// TIA Portal V20 export
TYPE "Udt_CarCode"
   STRUCT
      Plant_Identifier : WString[24];
      CarCode : Int;   // BadyCode
      Reserve1 : Int;
      Reserve2 : Int;
      Reserve3 : Int;
      Reserve4 : Int;
   END_STRUCT;
END_TYPE
